(* PLC project SupervisionStaging.project, CODESYS CODESYS V3.5 SP19 Patch 1 *)
(* stored: creationDateTime 2026-08-02T00:00:00, modificationDateTime 2026-08-02T00:00:00 *)

PROGRAM PRG_07_Supervision_CFC
  VAR
    instSupervisionProjection : FB_SupervisionProjection;
  END_VAR
  VAR_OUTPUT
    Ready : BOOL;
  END_VAR

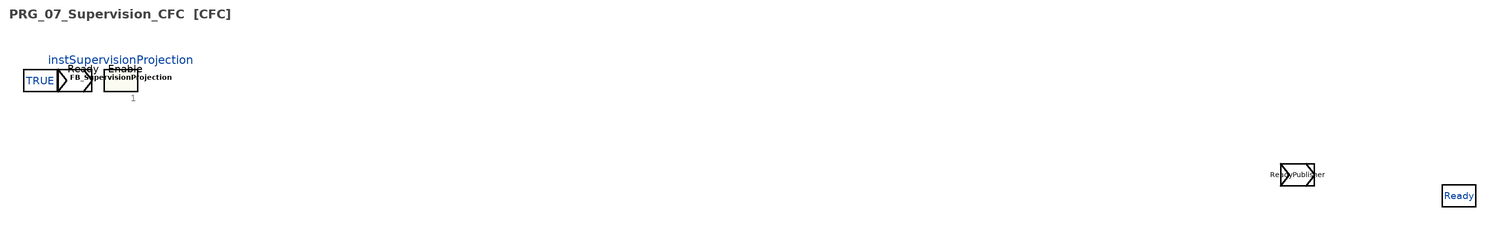
(* CFC diagram, written out as Structured Text *)
instSupervisionProjection(Enable := TRUE);
Ready := instSupervisionProjection.Ready;
END_PROGRAM
